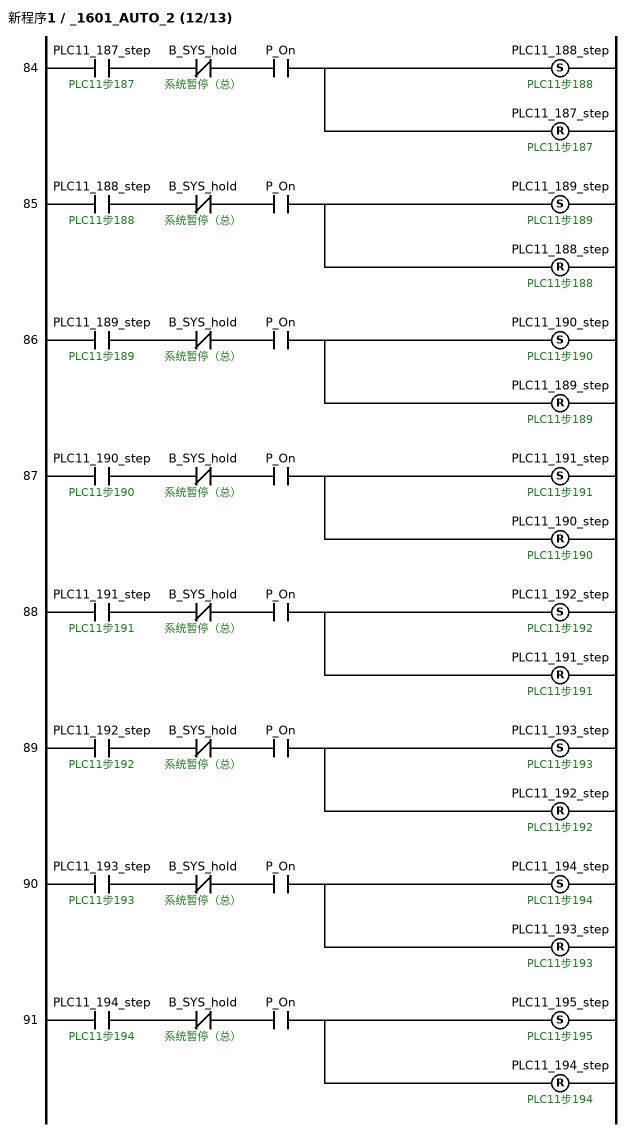
; [picture p48: 新程序1 / _1601_AUTO_2, rungs 84-91]
; rung 84
LD PLC11_187_step  ; PLC11步187
ANDNOT B_SYS_hold  ; 系统暂停（总）
AND P_On
SET PLC11_188_step  ; PLC11步188
RSET PLC11_187_step  ; PLC11步187
; rung 85
LD PLC11_188_step  ; PLC11步188
ANDNOT B_SYS_hold  ; 系统暂停（总）
AND P_On
SET PLC11_189_step  ; PLC11步189
RSET PLC11_188_step  ; PLC11步188
; rung 86
LD PLC11_189_step  ; PLC11步189
ANDNOT B_SYS_hold  ; 系统暂停（总）
AND P_On
SET PLC11_190_step  ; PLC11步190
RSET PLC11_189_step  ; PLC11步189
; rung 87
LD PLC11_190_step  ; PLC11步190
ANDNOT B_SYS_hold  ; 系统暂停（总）
AND P_On
SET PLC11_191_step  ; PLC11步191
RSET PLC11_190_step  ; PLC11步190
; rung 88
LD PLC11_191_step  ; PLC11步191
ANDNOT B_SYS_hold  ; 系统暂停（总）
AND P_On
SET PLC11_192_step  ; PLC11步192
RSET PLC11_191_step  ; PLC11步191
; rung 89
LD PLC11_192_step  ; PLC11步192
ANDNOT B_SYS_hold  ; 系统暂停（总）
AND P_On
SET PLC11_193_step  ; PLC11步193
RSET PLC11_192_step  ; PLC11步192
; rung 90
LD PLC11_193_step  ; PLC11步193
ANDNOT B_SYS_hold  ; 系统暂停（总）
AND P_On
SET PLC11_194_step  ; PLC11步194
RSET PLC11_193_step  ; PLC11步193
; rung 91
LD PLC11_194_step  ; PLC11步194
ANDNOT B_SYS_hold  ; 系统暂停（总）
AND P_On
SET PLC11_195_step  ; PLC11步195
RSET PLC11_194_step  ; PLC11步194

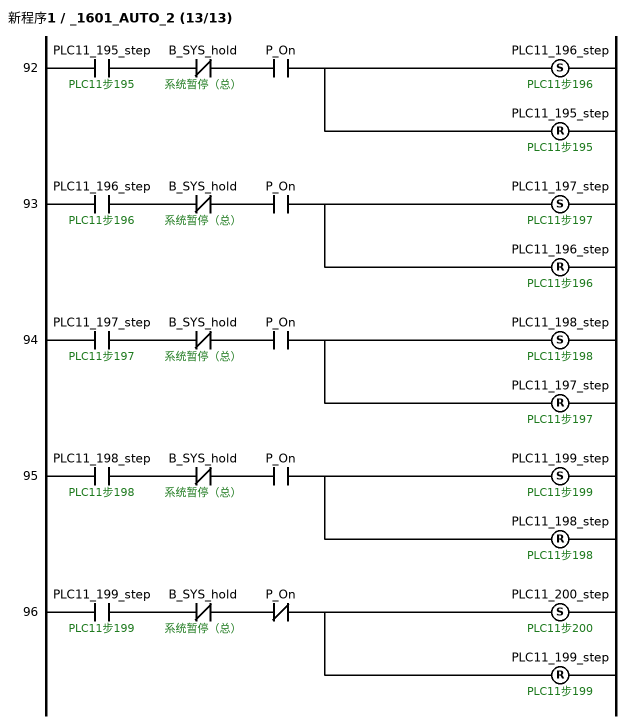
; rung 92
LD PLC11_195_step  ; PLC11步195
ANDNOT B_SYS_hold  ; 系统暂停（总）
AND P_On
SET PLC11_196_step  ; PLC11步196
RSET PLC11_195_step  ; PLC11步195
; rung 93
LD PLC11_196_step  ; PLC11步196
ANDNOT B_SYS_hold  ; 系统暂停（总）
AND P_On
SET PLC11_197_step  ; PLC11步197
RSET PLC11_196_step  ; PLC11步196
; rung 94
LD PLC11_197_step  ; PLC11步197
ANDNOT B_SYS_hold  ; 系统暂停（总）
AND P_On
SET PLC11_198_step  ; PLC11步198
RSET PLC11_197_step  ; PLC11步197
; rung 95
LD PLC11_198_step  ; PLC11步198
ANDNOT B_SYS_hold  ; 系统暂停（总）
AND P_On
SET PLC11_199_step  ; PLC11步199
RSET PLC11_198_step  ; PLC11步198
; rung 96
LD PLC11_199_step  ; PLC11步199
ANDNOT B_SYS_hold  ; 系统暂停（总）
ANDNOT P_On
SET PLC11_200_step  ; PLC11步200
RSET PLC11_199_step  ; PLC11步199

### Section _1601_AUTO_start

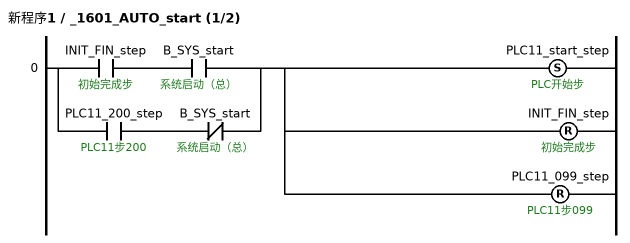
; rung 0
LD INIT_FIN_step  ; 初始完成步
AND B_SYS_start  ; 系统启动（总）
LD PLC11_200_step  ; PLC11步200
ANDNOT B_SYS_start  ; 系统启动（总）
ORLD
SET PLC11_start_step  ; PLC开始步
RSET INIT_FIN_step  ; 初始完成步
RSET PLC11_099_step  ; PLC11步099

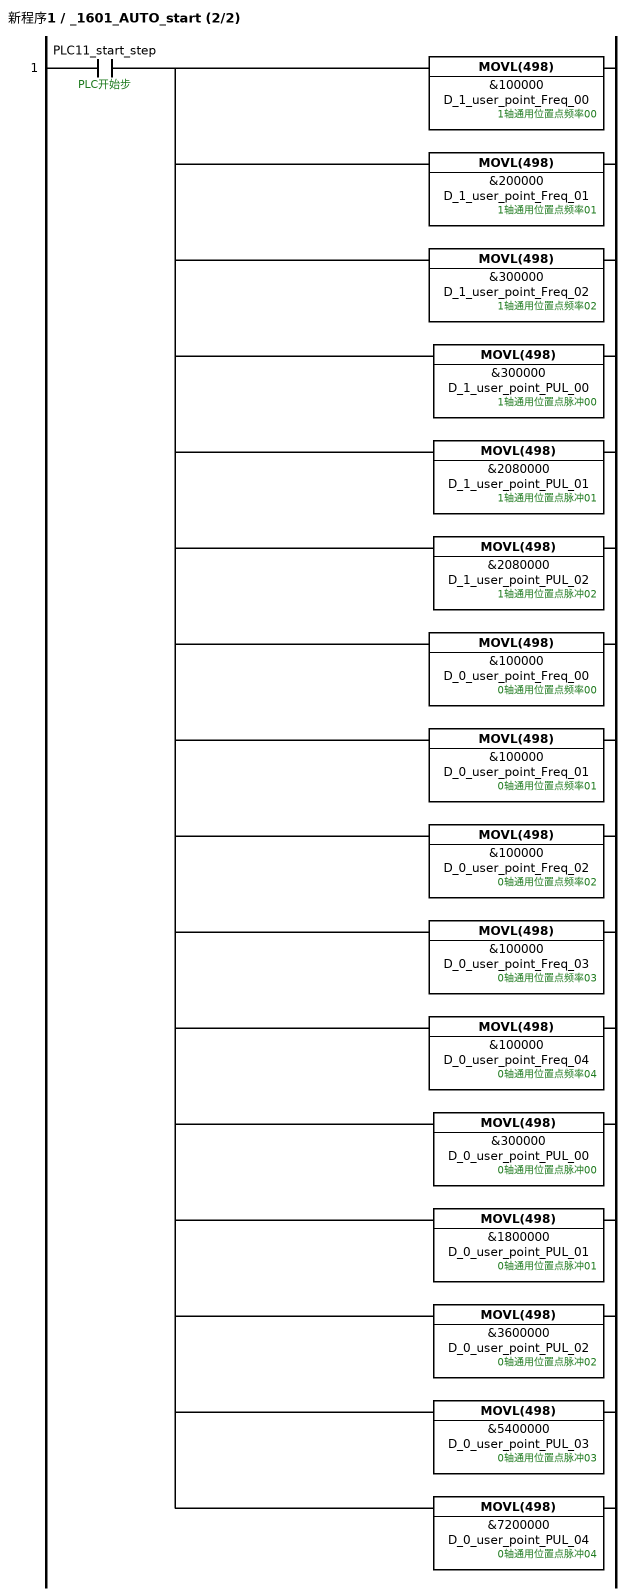
; rung 1
LD PLC11_start_step  ; PLC开始步
MOVL(498) &100000 D_1_user_point_Freq_00  ; 1轴通用位置点频率00
MOVL(498) &200000 D_1_user_point_Freq_01  ; 1轴通用位置点频率01
MOVL(498) &300000 D_1_user_point_Freq_02  ; 1轴通用位置点频率02
MOVL(498) &300000 D_1_user_point_PUL_00  ; 1轴通用位置点脉冲00
MOVL(498) &2080000 D_1_user_point_PUL_01  ; 1轴通用位置点脉冲01
MOVL(498) &2080000 D_1_user_point_PUL_02  ; 1轴通用位置点脉冲02
MOVL(498) &100000 D_0_user_point_Freq_00  ; 0轴通用位置点频率00
MOVL(498) &100000 D_0_user_point_Freq_01  ; 0轴通用位置点频率01
MOVL(498) &100000 D_0_user_point_Freq_02  ; 0轴通用位置点频率02
MOVL(498) &100000 D_0_user_point_Freq_03  ; 0轴通用位置点频率03
MOVL(498) &100000 D_0_user_point_Freq_04  ; 0轴通用位置点频率04
MOVL(498) &300000 D_0_user_point_PUL_00  ; 0轴通用位置点脉冲00
MOVL(498) &1800000 D_0_user_point_PUL_01  ; 0轴通用位置点脉冲01
MOVL(498) &3600000 D_0_user_point_PUL_02  ; 0轴通用位置点脉冲02
MOVL(498) &5400000 D_0_user_point_PUL_03  ; 0轴通用位置点脉冲03
MOVL(498) &7200000 D_0_user_point_PUL_04  ; 0轴通用位置点脉冲04

### Section _1601_AUTO_stop

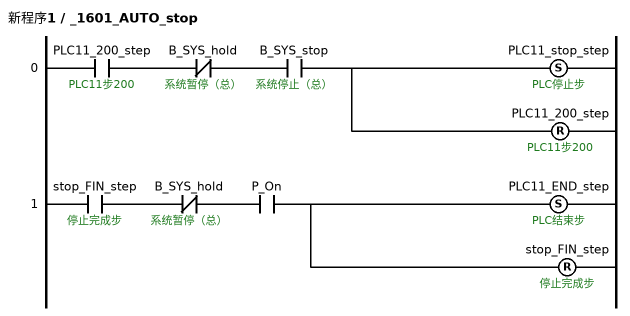
; rung 0
LD PLC11_200_step  ; PLC11步200
ANDNOT B_SYS_hold  ; 系统暂停（总）
AND B_SYS_stop  ; 系统停止（总）
SET PLC11_stop_step  ; PLC停止步
RSET PLC11_200_step  ; PLC11步200
; rung 1
LD stop_FIN_step  ; 停止完成步
ANDNOT B_SYS_hold  ; 系统暂停（总）
AND P_On
SET PLC11_END_step  ; PLC结束步
RSET stop_FIN_step  ; 停止完成步

### Section _1601_INIT

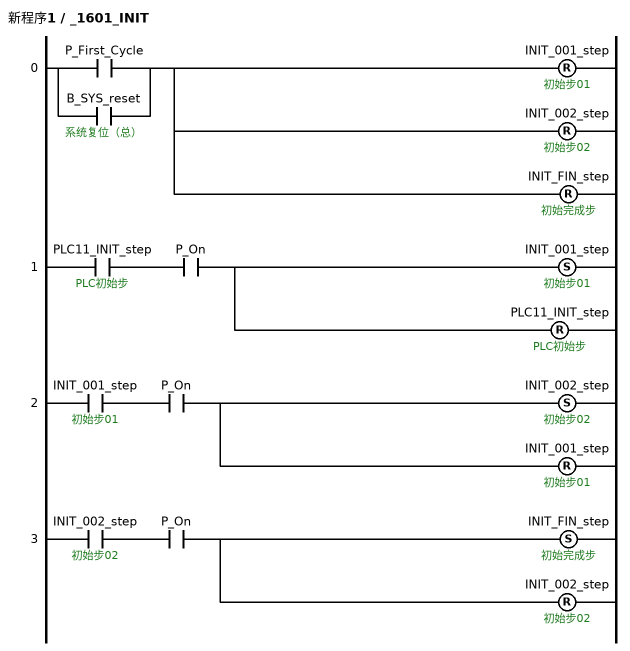
; rung 0
LD P_First_Cycle
OR B_SYS_reset  ; 系统复位（总）
RSET INIT_001_step  ; 初始步01
RSET INIT_002_step  ; 初始步02
RSET INIT_FIN_step  ; 初始完成步
; rung 1
LD PLC11_INIT_step  ; PLC初始步
AND P_On
SET INIT_001_step  ; 初始步01
RSET PLC11_INIT_step  ; PLC初始步
; rung 2
LD INIT_001_step  ; 初始步01
AND P_On
SET INIT_002_step  ; 初始步02
RSET INIT_001_step  ; 初始步01
; rung 3
LD INIT_002_step  ; 初始步02
AND P_On
SET INIT_FIN_step  ; 初始完成步
RSET INIT_002_step  ; 初始步02

### Section _1601_start

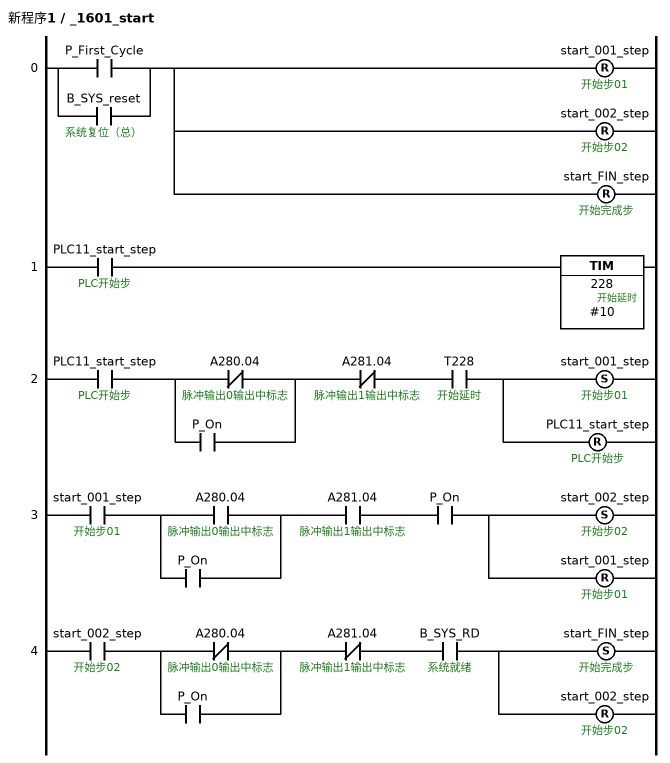
; rung 0
LD P_First_Cycle
OR B_SYS_reset  ; 系统复位（总）
RSET start_001_step  ; 开始步01
RSET start_002_step  ; 开始步02
RSET start_FIN_step  ; 开始完成步
; rung 1
LD PLC11_start_step  ; PLC开始步
TIM 228 #10  ; 开始延时
; rung 2
LD PLC11_start_step  ; PLC开始步
LDNOT A280.04  ; 脉冲输出0输出中标志
OR P_On
ANDLD
ANDNOT A281.04  ; 脉冲输出1输出中标志
AND T228  ; 开始延时
SET start_001_step  ; 开始步01
RSET PLC11_start_step  ; PLC开始步
; rung 3
LD start_001_step  ; 开始步01
LD A280.04  ; 脉冲输出0输出中标志
OR P_On
ANDLD
AND A281.04  ; 脉冲输出1输出中标志
AND P_On
SET start_002_step  ; 开始步02
RSET start_001_step  ; 开始步01
; rung 4
LD start_002_step  ; 开始步02
LDNOT A280.04  ; 脉冲输出0输出中标志
OR P_On
ANDLD
ANDNOT A281.04  ; 脉冲输出1输出中标志
AND B_SYS_RD  ; 系统就绪
SET start_FIN_step  ; 开始完成步
RSET start_002_step  ; 开始步02

### Section _1601_stop

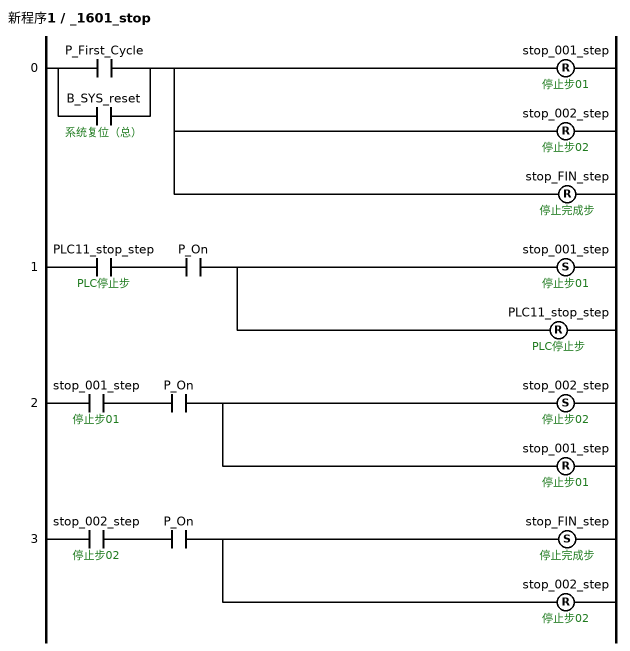
; rung 0
LD P_First_Cycle
OR B_SYS_reset  ; 系统复位（总）
RSET stop_001_step  ; 停止步01
RSET stop_002_step  ; 停止步02
RSET stop_FIN_step  ; 停止完成步
; rung 1
LD PLC11_stop_step  ; PLC停止步
AND P_On
SET stop_001_step  ; 停止步01
RSET PLC11_stop_step  ; PLC停止步
; rung 2
LD stop_001_step  ; 停止步01
AND P_On
SET stop_002_step  ; 停止步02
RSET stop_001_step  ; 停止步01
; rung 3
LD stop_002_step  ; 停止步02
AND P_On
SET stop_FIN_step  ; 停止完成步
RSET stop_002_step  ; 停止步02

### Section _1601_ERR

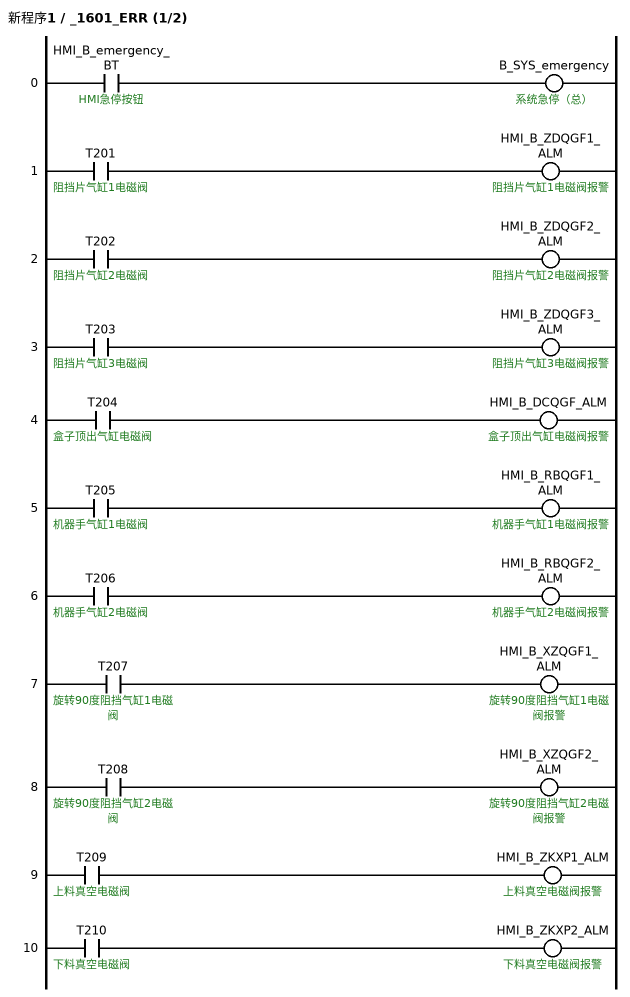
; rung 0
LD HMI_B_emergency_BT  ; HMI急停按钮
OUT B_SYS_emergency  ; 系统急停（总）
; rung 1
LD T201  ; 阻挡片气缸1电磁阀
OUT HMI_B_ZDQGF1_ALM  ; 阻挡片气缸1电磁阀报警
; rung 2
LD T202  ; 阻挡片气缸2电磁阀
OUT HMI_B_ZDQGF2_ALM  ; 阻挡片气缸2电磁阀报警
; rung 3
LD T203  ; 阻挡片气缸3电磁阀
OUT HMI_B_ZDQGF3_ALM  ; 阻挡片气缸3电磁阀报警
; rung 4
LD T204  ; 盒子顶出气缸电磁阀
OUT HMI_B_DCQGF_ALM  ; 盒子顶出气缸电磁阀报警
; rung 5
LD T205  ; 机器手气缸1电磁阀
OUT HMI_B_RBQGF1_ALM  ; 机器手气缸1电磁阀报警
; rung 6
LD T206  ; 机器手气缸2电磁阀
OUT HMI_B_RBQGF2_ALM  ; 机器手气缸2电磁阀报警
; rung 7
LD T207  ; 旋转90度阻挡气缸1电磁阀
OUT HMI_B_XZQGF1_ALM  ; 旋转90度阻挡气缸1电磁阀报警
; rung 8
LD T208  ; 旋转90度阻挡气缸2电磁阀
OUT HMI_B_XZQGF2_ALM  ; 旋转90度阻挡气缸2电磁阀报警
; rung 9
LD T209  ; 上料真空电磁阀
OUT HMI_B_ZKXP1_ALM  ; 上料真空电磁阀报警
; rung 10
LD T210  ; 下料真空电磁阀
OUT HMI_B_ZKXP2_ALM  ; 下料真空电磁阀报警

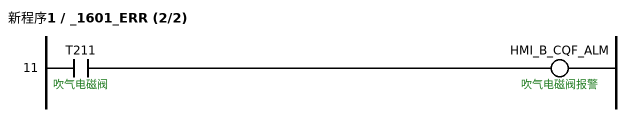
; rung 11
LD T211  ; 吹气电磁阀
OUT HMI_B_CQF_ALM  ; 吹气电磁阀报警

### Section SERVO_INIT

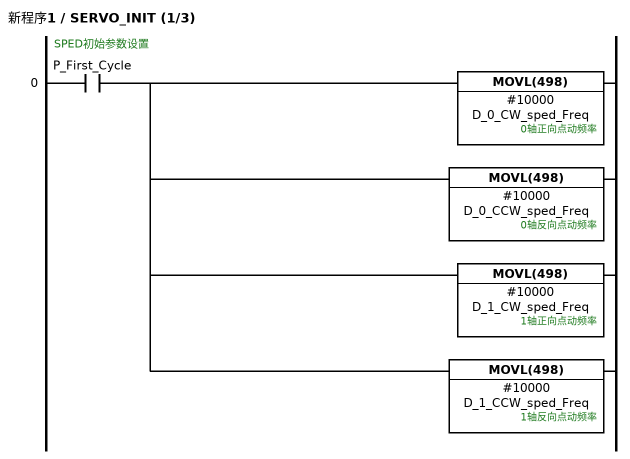
; rung 0: SPED初始参数设置
LD P_First_Cycle
MOVL(498) #10000 D_0_CW_sped_Freq  ; 0轴正向点动频率
MOVL(498) #10000 D_0_CCW_sped_Freq  ; 0轴反向点动频率
MOVL(498) #10000 D_1_CW_sped_Freq  ; 1轴正向点动频率
MOVL(498) #10000 D_1_CCW_sped_Freq  ; 1轴反向点动频率

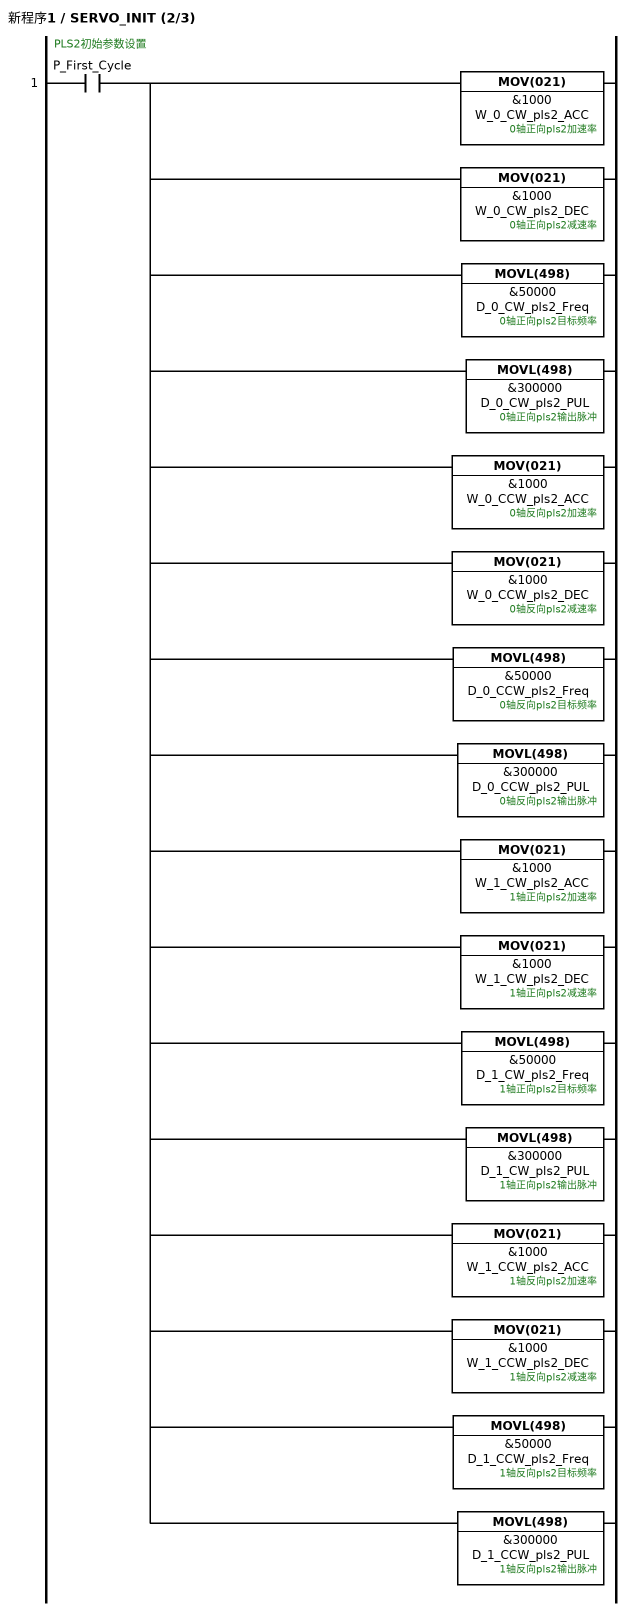
; rung 1: PLS2初始参数设置
LD P_First_Cycle
MOV(021) &1000 W_0_CW_pls2_ACC  ; 0轴正向pls2加速率
MOV(021) &1000 W_0_CW_pls2_DEC  ; 0轴正向pls2减速率
MOVL(498) &50000 D_0_CW_pls2_Freq  ; 0轴正向pls2目标频率
MOVL(498) &300000 D_0_CW_pls2_PUL  ; 0轴正向pls2输出脉冲
MOV(021) &1000 W_0_CCW_pls2_ACC  ; 0轴反向pls2加速率
MOV(021) &1000 W_0_CCW_pls2_DEC  ; 0轴反向pls2减速率
MOVL(498) &50000 D_0_CCW_pls2_Freq  ; 0轴反向pls2目标频率
MOVL(498) &300000 D_0_CCW_pls2_PUL  ; 0轴反向pls2输出脉冲
MOV(021) &1000 W_1_CW_pls2_ACC  ; 1轴正向pls2加速率
MOV(021) &1000 W_1_CW_pls2_DEC  ; 1轴正向pls2减速率
MOVL(498) &50000 D_1_CW_pls2_Freq  ; 1轴正向pls2目标频率
MOVL(498) &300000 D_1_CW_pls2_PUL  ; 1轴正向pls2输出脉冲
MOV(021) &1000 W_1_CCW_pls2_ACC  ; 1轴反向pls2加速率
MOV(021) &1000 W_1_CCW_pls2_DEC  ; 1轴反向pls2减速率
MOVL(498) &50000 D_1_CCW_pls2_Freq  ; 1轴反向pls2目标频率
MOVL(498) &300000 D_1_CCW_pls2_PUL  ; 1轴反向pls2输出脉冲

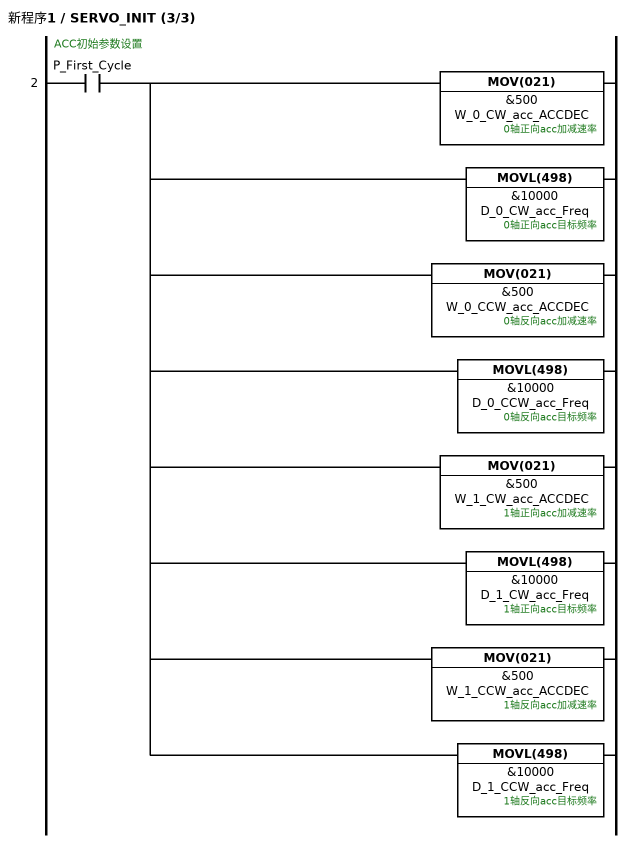
; rung 2: ACC初始参数设置
LD P_First_Cycle
MOV(021) &500 W_0_CW_acc_ACCDEC  ; 0轴正向acc加减速率
MOVL(498) &10000 D_0_CW_acc_Freq  ; 0轴正向acc目标频率
MOV(021) &500 W_0_CCW_acc_ACCDEC  ; 0轴反向acc加减速率
MOVL(498) &10000 D_0_CCW_acc_Freq  ; 0轴反向acc目标频率
MOV(021) &500 W_1_CW_acc_ACCDEC  ; 1轴正向acc加减速率
MOVL(498) &10000 D_1_CW_acc_Freq  ; 1轴正向acc目标频率
MOV(021) &500 W_1_CCW_acc_ACCDEC  ; 1轴反向acc加减速率
MOVL(498) &10000 D_1_CCW_acc_Freq  ; 1轴反向acc目标频率

### Section SERVO_JOG

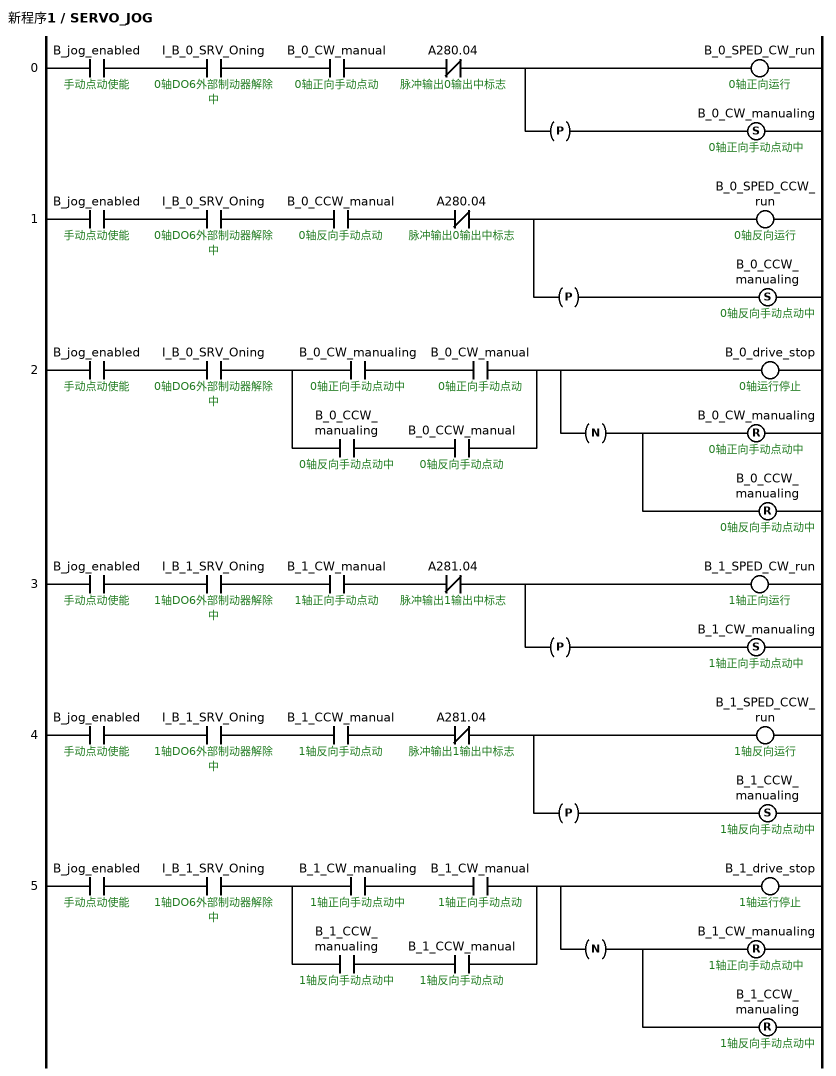
; rung 0
LD B_jog_enabled  ; 手动点动使能
AND I_B_0_SRV_Oning  ; 0轴DO6外部制动器解除中
AND B_0_CW_manual  ; 0轴正向手动点动
ANDNOT A280.04  ; 脉冲输出0输出中标志
OUT B_0_SPED_CW_run  ; 0轴正向运行
UP(521)
SET B_0_CW_manualing  ; 0轴正向手动点动中
; rung 1
LD B_jog_enabled  ; 手动点动使能
AND I_B_0_SRV_Oning  ; 0轴DO6外部制动器解除中
AND B_0_CCW_manual  ; 0轴反向手动点动
ANDNOT A280.04  ; 脉冲输出0输出中标志
OUT B_0_SPED_CCW_run  ; 0轴反向运行
UP(521)
SET B_0_CCW_manualing  ; 0轴反向手动点动中
; rung 2
LD B_jog_enabled  ; 手动点动使能
AND I_B_0_SRV_Oning  ; 0轴DO6外部制动器解除中
LD B_0_CW_manualing  ; 0轴正向手动点动中
AND B_0_CW_manual  ; 0轴正向手动点动
LD B_0_CCW_manualing  ; 0轴反向手动点动中
AND B_0_CCW_manual  ; 0轴反向手动点动
ORLD
ANDLD
OUT B_0_drive_stop  ; 0轴运行停止
DOWN(522)
RSET B_0_CW_manualing  ; 0轴正向手动点动中
RSET B_0_CCW_manualing  ; 0轴反向手动点动中
; rung 3
LD B_jog_enabled  ; 手动点动使能
AND I_B_1_SRV_Oning  ; 1轴DO6外部制动器解除中
AND B_1_CW_manual  ; 1轴正向手动点动
ANDNOT A281.04  ; 脉冲输出1输出中标志
OUT B_1_SPED_CW_run  ; 1轴正向运行
UP(521)
SET B_1_CW_manualing  ; 1轴正向手动点动中
; rung 4
LD B_jog_enabled  ; 手动点动使能
AND I_B_1_SRV_Oning  ; 1轴DO6外部制动器解除中
AND B_1_CCW_manual  ; 1轴反向手动点动
ANDNOT A281.04  ; 脉冲输出1输出中标志
OUT B_1_SPED_CCW_run  ; 1轴反向运行
UP(521)
SET B_1_CCW_manualing  ; 1轴反向手动点动中
; rung 5
LD B_jog_enabled  ; 手动点动使能
AND I_B_1_SRV_Oning  ; 1轴DO6外部制动器解除中
LD B_1_CW_manualing  ; 1轴正向手动点动中
AND B_1_CW_manual  ; 1轴正向手动点动
LD B_1_CCW_manualing  ; 1轴反向手动点动中
AND B_1_CCW_manual  ; 1轴反向手动点动
ORLD
ANDLD
OUT B_1_drive_stop  ; 1轴运行停止
DOWN(522)
RSET B_1_CW_manualing  ; 1轴正向手动点动中
RSET B_1_CCW_manualing  ; 1轴反向手动点动中

### Section SERVO_IO

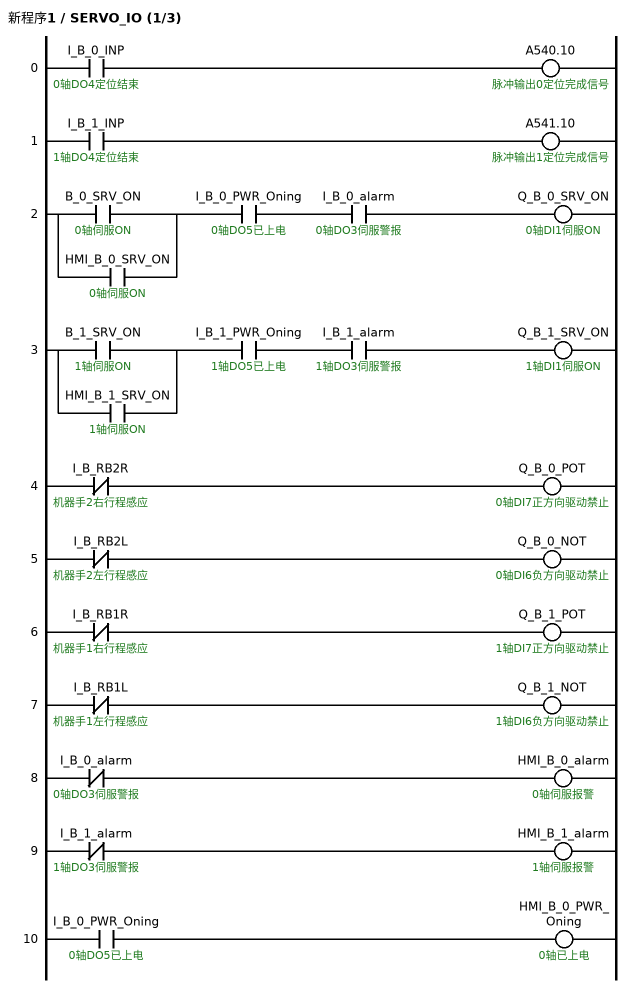
; rung 0
LD I_B_0_INP  ; 0轴DO4定位结束
OUT A540.10  ; 脉冲输出0定位完成信号
; rung 1
LD I_B_1_INP  ; 1轴DO4定位结束
OUT A541.10  ; 脉冲输出1定位完成信号
; rung 2
LD B_0_SRV_ON  ; 0轴伺服ON
OR HMI_B_0_SRV_ON  ; 0轴伺服ON
AND I_B_0_PWR_Oning  ; 0轴DO5已上电
AND I_B_0_alarm  ; 0轴DO3伺服警报
OUT Q_B_0_SRV_ON  ; 0轴DI1伺服ON
; rung 3
LD B_1_SRV_ON  ; 1轴伺服ON
OR HMI_B_1_SRV_ON  ; 1轴伺服ON
AND I_B_1_PWR_Oning  ; 1轴DO5已上电
AND I_B_1_alarm  ; 1轴DO3伺服警报
OUT Q_B_1_SRV_ON  ; 1轴DI1伺服ON
; rung 4
LDNOT I_B_RB2R  ; 机器手2右行程感应
OUT Q_B_0_POT  ; 0轴DI7正方向驱动禁止
; rung 5
LDNOT I_B_RB2L  ; 机器手2左行程感应
OUT Q_B_0_NOT  ; 0轴DI6负方向驱动禁止
; rung 6
LDNOT I_B_RB1R  ; 机器手1右行程感应
OUT Q_B_1_POT  ; 1轴DI7正方向驱动禁止
; rung 7
LDNOT I_B_RB1L  ; 机器手1左行程感应
OUT Q_B_1_NOT  ; 1轴DI6负方向驱动禁止
; rung 8
LDNOT I_B_0_alarm  ; 0轴DO3伺服警报
OUT HMI_B_0_alarm  ; 0轴伺服报警
; rung 9
LDNOT I_B_1_alarm  ; 1轴DO3伺服警报
OUT HMI_B_1_alarm  ; 1轴伺服报警
; rung 10
LD I_B_0_PWR_Oning  ; 0轴DO5已上电
OUT HMI_B_0_PWR_Oning  ; 0轴已上电

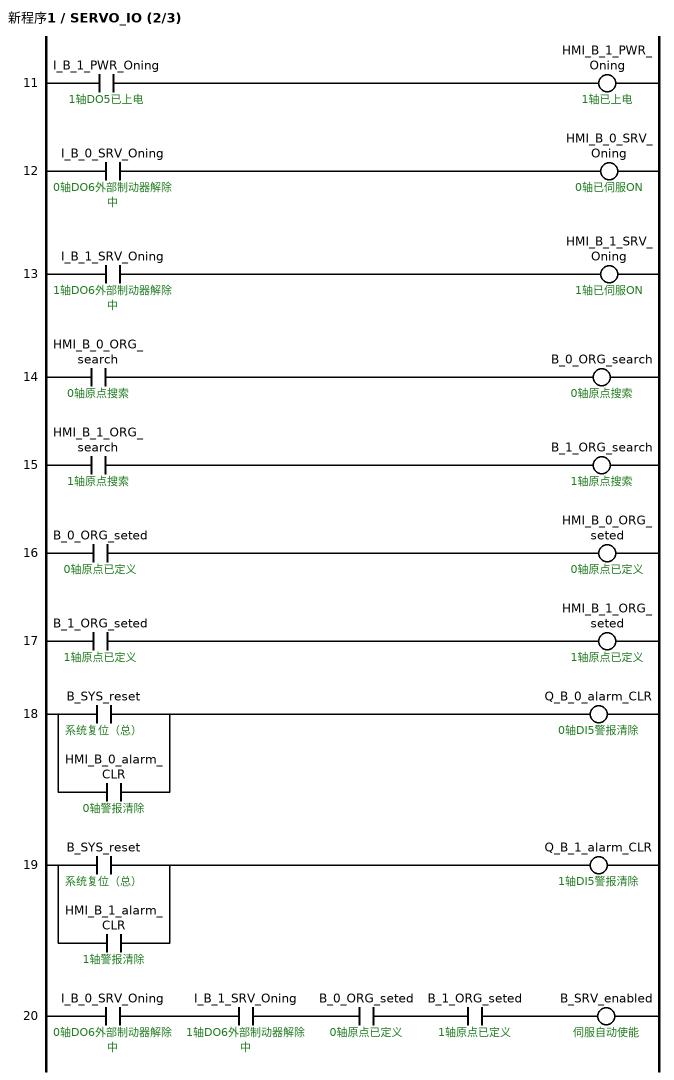
; rung 11
LD I_B_1_PWR_Oning  ; 1轴DO5已上电
OUT HMI_B_1_PWR_Oning  ; 1轴已上电
; rung 12
LD I_B_0_SRV_Oning  ; 0轴DO6外部制动器解除中
OUT HMI_B_0_SRV_Oning  ; 0轴已伺服ON
; rung 13
LD I_B_1_SRV_Oning  ; 1轴DO6外部制动器解除中
OUT HMI_B_1_SRV_Oning  ; 1轴已伺服ON
; rung 14
LD HMI_B_0_ORG_search  ; 0轴原点搜索
OUT B_0_ORG_search  ; 0轴原点搜索
; rung 15
LD HMI_B_1_ORG_search  ; 1轴原点搜索
OUT B_1_ORG_search  ; 1轴原点搜索
; rung 16
LD B_0_ORG_seted  ; 0轴原点已定义
OUT HMI_B_0_ORG_seted  ; 0轴原点已定义
; rung 17
LD B_1_ORG_seted  ; 1轴原点已定义
OUT HMI_B_1_ORG_seted  ; 1轴原点已定义
; rung 18
LD B_SYS_reset  ; 系统复位（总）
OR HMI_B_0_alarm_CLR  ; 0轴警报清除
OUT Q_B_0_alarm_CLR  ; 0轴DI5警报清除
; rung 19
LD B_SYS_reset  ; 系统复位（总）
OR HMI_B_1_alarm_CLR  ; 1轴警报清除
OUT Q_B_1_alarm_CLR  ; 1轴DI5警报清除
; rung 20
LD I_B_0_SRV_Oning  ; 0轴DO6外部制动器解除中
AND I_B_1_SRV_Oning  ; 1轴DO6外部制动器解除中
AND B_0_ORG_seted  ; 0轴原点已定义
AND B_1_ORG_seted  ; 1轴原点已定义
OUT B_SRV_enabled  ; 伺服自动使能

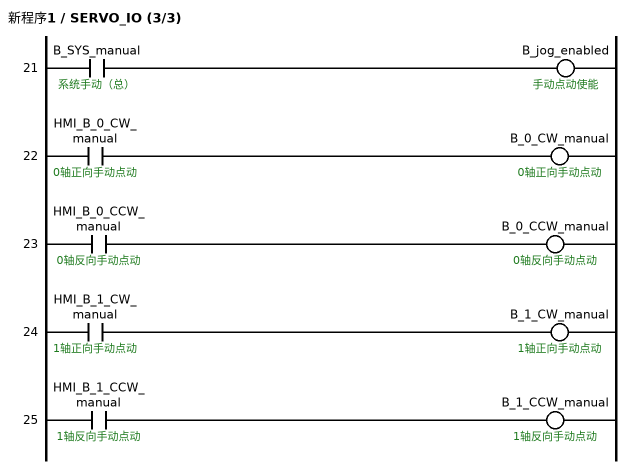
; rung 21
LD B_SYS_manual  ; 系统手动（总）
OUT B_jog_enabled  ; 手动点动使能
; rung 22
LD HMI_B_0_CW_manual  ; 0轴正向手动点动
OUT B_0_CW_manual  ; 0轴正向手动点动
; rung 23
LD HMI_B_0_CCW_manual  ; 0轴反向手动点动
OUT B_0_CCW_manual  ; 0轴反向手动点动
; rung 24
LD HMI_B_1_CW_manual  ; 1轴正向手动点动
OUT B_1_CW_manual  ; 1轴正向手动点动
; rung 25
LD HMI_B_1_CCW_manual  ; 1轴反向手动点动
OUT B_1_CCW_manual  ; 1轴反向手动点动

### Section SERVO

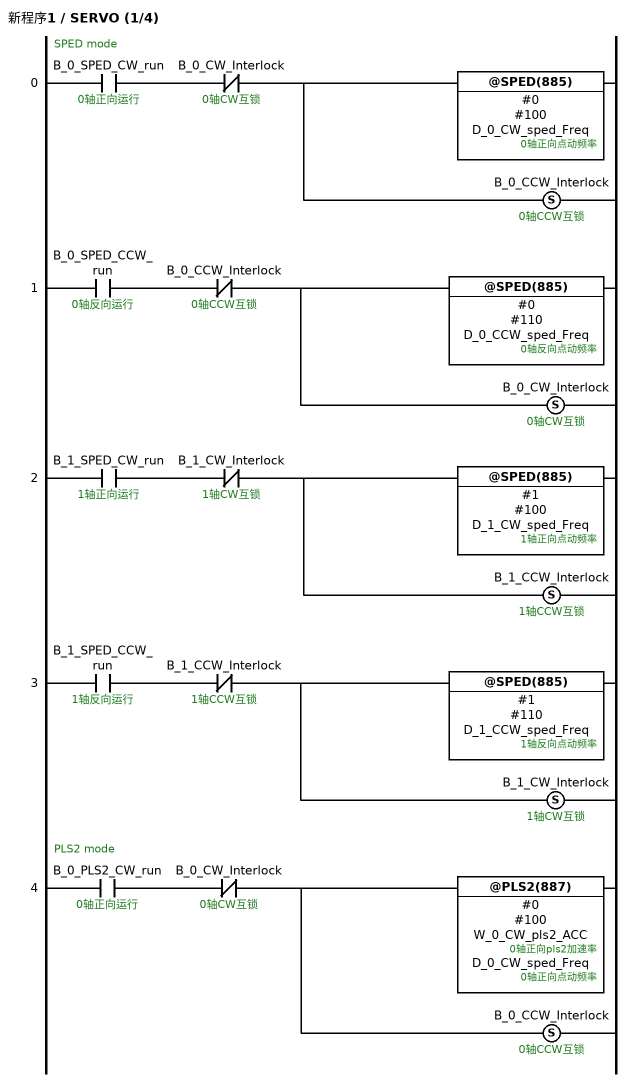
; rung 0: SPED mode
LD B_0_SPED_CW_run  ; 0轴正向运行
ANDNOT B_0_CW_Interlock  ; 0轴CW互锁
@SPED(885) #0 #100 D_0_CW_sped_Freq  ; 0轴正向点动频率
SET B_0_CCW_Interlock  ; 0轴CCW互锁
; rung 1
LD B_0_SPED_CCW_run  ; 0轴反向运行
ANDNOT B_0_CCW_Interlock  ; 0轴CCW互锁
@SPED(885) #0 #110 D_0_CCW_sped_Freq  ; 0轴反向点动频率
SET B_0_CW_Interlock  ; 0轴CW互锁
; rung 2
LD B_1_SPED_CW_run  ; 1轴正向运行
ANDNOT B_1_CW_Interlock  ; 1轴CW互锁
@SPED(885) #1 #100 D_1_CW_sped_Freq  ; 1轴正向点动频率
SET B_1_CCW_Interlock  ; 1轴CCW互锁
; rung 3
LD B_1_SPED_CCW_run  ; 1轴反向运行
ANDNOT B_1_CCW_Interlock  ; 1轴CCW互锁
@SPED(885) #1 #110 D_1_CCW_sped_Freq  ; 1轴反向点动频率
SET B_1_CW_Interlock  ; 1轴CW互锁
; rung 4: PLS2 mode
LD B_0_PLS2_CW_run  ; 0轴正向运行
ANDNOT B_0_CW_Interlock  ; 0轴CW互锁
@PLS2(887) #0 #100 W_0_CW_pls2_ACC D_0_CW_sped_Freq  ; 0轴正向pls2加速率, 0轴正向点动频率
SET B_0_CCW_Interlock  ; 0轴CCW互锁

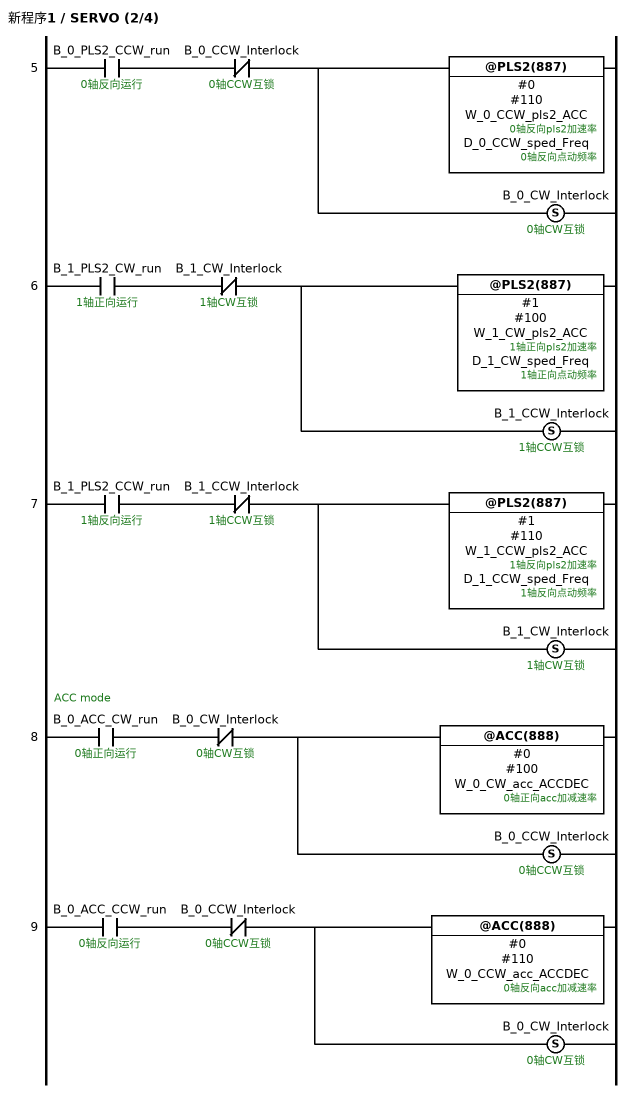
; rung 5
LD B_0_PLS2_CCW_run  ; 0轴反向运行
ANDNOT B_0_CCW_Interlock  ; 0轴CCW互锁
@PLS2(887) #0 #110 W_0_CCW_pls2_ACC D_0_CCW_sped_Freq  ; 0轴反向pls2加速率, 0轴反向点动频率
SET B_0_CW_Interlock  ; 0轴CW互锁
; rung 6
LD B_1_PLS2_CW_run  ; 1轴正向运行
ANDNOT B_1_CW_Interlock  ; 1轴CW互锁
@PLS2(887) #1 #100 W_1_CW_pls2_ACC D_1_CW_sped_Freq  ; 1轴正向pls2加速率, 1轴正向点动频率
SET B_1_CCW_Interlock  ; 1轴CCW互锁
; rung 7
LD B_1_PLS2_CCW_run  ; 1轴反向运行
ANDNOT B_1_CCW_Interlock  ; 1轴CCW互锁
@PLS2(887) #1 #110 W_1_CCW_pls2_ACC D_1_CCW_sped_Freq  ; 1轴反向pls2加速率, 1轴反向点动频率
SET B_1_CW_Interlock  ; 1轴CW互锁
; rung 8: ACC mode
LD B_0_ACC_CW_run  ; 0轴正向运行
ANDNOT B_0_CW_Interlock  ; 0轴CW互锁
@ACC(888) #0 #100 W_0_CW_acc_ACCDEC  ; 0轴正向acc加减速率
SET B_0_CCW_Interlock  ; 0轴CCW互锁
; rung 9
LD B_0_ACC_CCW_run  ; 0轴反向运行
ANDNOT B_0_CCW_Interlock  ; 0轴CCW互锁
@ACC(888) #0 #110 W_0_CCW_acc_ACCDEC  ; 0轴反向acc加减速率
SET B_0_CW_Interlock  ; 0轴CW互锁

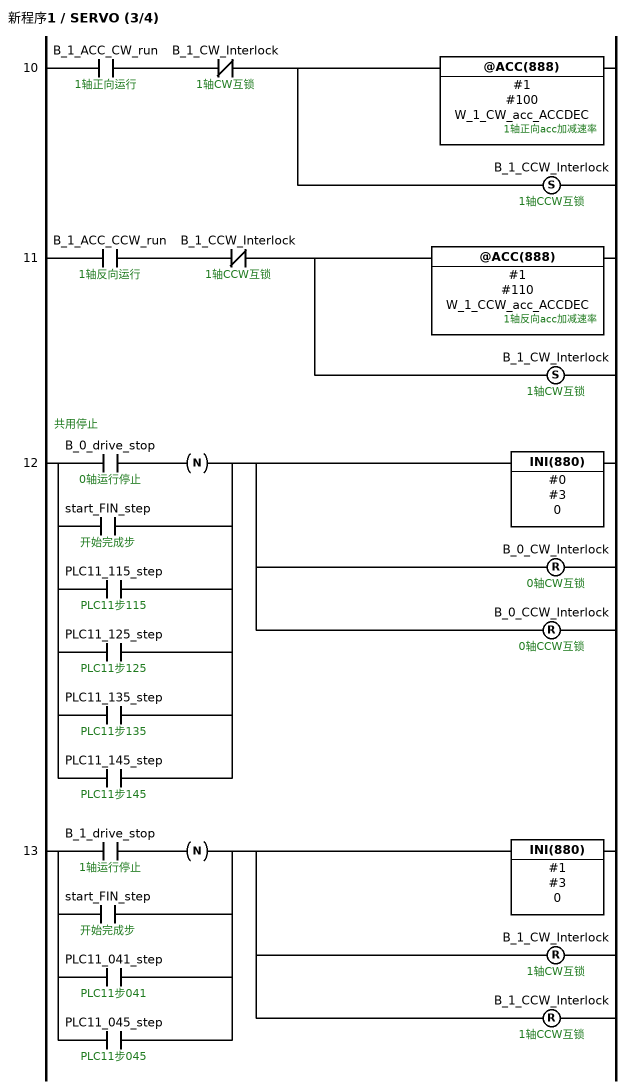
; rung 10
LD B_1_ACC_CW_run  ; 1轴正向运行
ANDNOT B_1_CW_Interlock  ; 1轴CW互锁
@ACC(888) #1 #100 W_1_CW_acc_ACCDEC  ; 1轴正向acc加减速率
SET B_1_CCW_Interlock  ; 1轴CCW互锁
; rung 11
LD B_1_ACC_CCW_run  ; 1轴反向运行
ANDNOT B_1_CCW_Interlock  ; 1轴CCW互锁
@ACC(888) #1 #110 W_1_CCW_acc_ACCDEC  ; 1轴反向acc加减速率
SET B_1_CW_Interlock  ; 1轴CW互锁
; rung 12: 共用停止
LD B_0_drive_stop  ; 0轴运行停止
DOWN(522)
OR start_FIN_step  ; 开始完成步
OR PLC11_115_step  ; PLC11步115
OR PLC11_125_step  ; PLC11步125
OR PLC11_135_step  ; PLC11步135
OR PLC11_145_step  ; PLC11步145
INI(880) #0 #3 0
RSET B_0_CW_Interlock  ; 0轴CW互锁
RSET B_0_CCW_Interlock  ; 0轴CCW互锁
; rung 13
LD B_1_drive_stop  ; 1轴运行停止
DOWN(522)
OR start_FIN_step  ; 开始完成步
OR PLC11_041_step  ; PLC11步041
OR PLC11_045_step  ; PLC11步045
INI(880) #1 #3 0
RSET B_1_CW_Interlock  ; 1轴CW互锁
RSET B_1_CCW_Interlock  ; 1轴CCW互锁

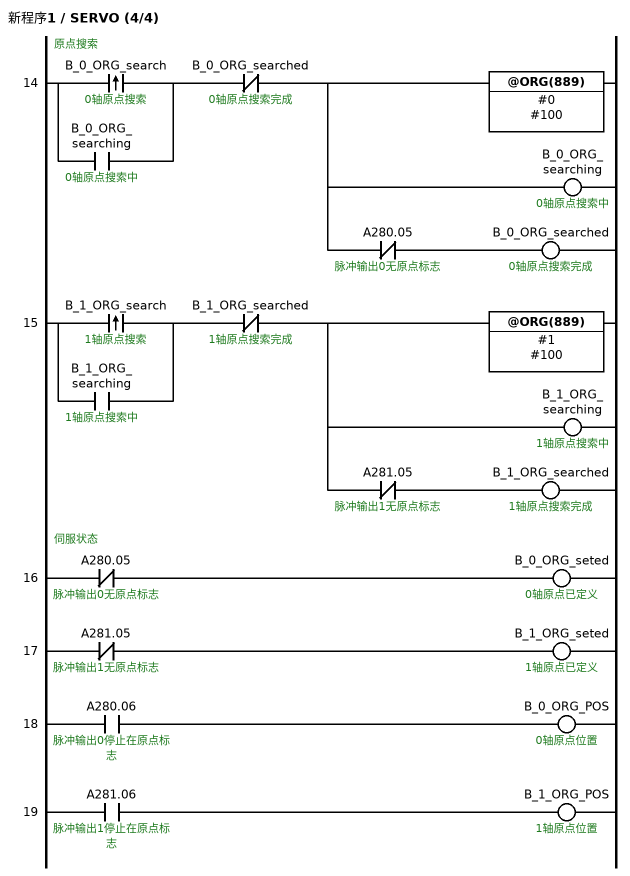
; rung 14: 原点搜索
@LD B_0_ORG_search  ; 0轴原点搜索
OR B_0_ORG_searching  ; 0轴原点搜索中
ANDNOT B_0_ORG_searched  ; 0轴原点搜索完成
@ORG(889) #0 #100
OUT B_0_ORG_searching  ; 0轴原点搜索中
ANDNOT A280.05  ; 脉冲输出0无原点标志
OUT B_0_ORG_searched  ; 0轴原点搜索完成
; rung 15
@LD B_1_ORG_search  ; 1轴原点搜索
OR B_1_ORG_searching  ; 1轴原点搜索中
ANDNOT B_1_ORG_searched  ; 1轴原点搜索完成
@ORG(889) #1 #100
OUT B_1_ORG_searching  ; 1轴原点搜索中
ANDNOT A281.05  ; 脉冲输出1无原点标志
OUT B_1_ORG_searched  ; 1轴原点搜索完成
; rung 16: 伺服状态
LDNOT A280.05  ; 脉冲输出0无原点标志
OUT B_0_ORG_seted  ; 0轴原点已定义
; rung 17
LDNOT A281.05  ; 脉冲输出1无原点标志
OUT B_1_ORG_seted  ; 1轴原点已定义
; rung 18
LD A280.06  ; 脉冲输出0停止在原点标志
OUT B_0_ORG_POS  ; 0轴原点位置
; rung 19
LD A281.06  ; 脉冲输出1停止在原点标志
OUT B_1_ORG_POS  ; 1轴原点位置

### Section END
; rung 0
END(001)